TYPE aT_Fan :
STRUCT
	SetSpeed: LREAL;
	PowerPercent: LREAL;
END_STRUCT
END_TYPE

(* stored: Version 1.1.0.1, ProductVersion 3.1.4024.4
   DUT aT_Fan: Id {c74f2963-2c8d-4521-87c4-922fa137d7e0} *)
